// TIA Portal V16 export
// export: Created 2024-09-05T17:39:25.2176429Z, ExportSetting WithDefaults, DisplayName Totally Integrated Automation Portal, DisplayVersion V16 Update 6, DisplayName TIA Portal Version Control Interface, DisplayVersion V16 Update 2, DisplayName TIA Portal Openness, DisplayVersion V16 Update 6, DisplayName STEP 7 Professional, DisplayVersion V16 Update 6, DisplayName STEP 7 Safety, DisplayVersion V16, DisplayName WinCC Advanced, DisplayVersion V16 Update 6
DATA_BLOCK "DB_DMC_string"   // DB2010
{ S7_Optimized_Access := 'TRUE' }
VERSION : 0.1
// stored: AutoNumber false, DBAccessibleFromOPCUA true, IsOnlyStoredInLoadMemory false, IsRetainMemResEnabled false, IsWriteProtectedInAS false, MemoryReserve 100
   VAR
      Extract_ST1 : Array[1..10] of String[25];
      Extract_ST2 : Array[1..10] of String[25];
      Concantenate_Wtring_ST1 : WString;
      Concantenate_Wtring_ST2 : WString;
      string_empty_st1 : Bool;
      string_empty_st2 : Bool;
   END_VAR
BEGIN
END_DATA_BLOCK
